FUNCTION_BLOCK FB_SimulatedScale EXTENDS FB_ComponentBase IMPLEMENTS I_Scale
VAR_INPUT
END_VAR
VAR_OUTPUT
END_VAR
VAR
END_VAR

{warning 'Add method implementation '}
METHOD CyclicLogic
END_METHOD

{warning 'Add method implementation '}
METHOD Tare
END_METHOD

{warning 'Add property implementation'}
PROPERTY Weight : LREAL
GET
END_GET
SET
END_SET
END_PROPERTY

END_FUNCTION_BLOCK

(* stored: Version 1.1.0.1
   POU FB_SimulatedScale: Id {4daf688a-6a4f-43ef-98c9-d12265253220}, SpecialFunc None
   Method CyclicLogic: Id {8eb76a38-87f9-4e72-b49b-7fc2f5b7cd9a}
   Method Tare: Id {bd2a2a9b-4af6-4061-af68-9126198b4727}
   Property Weight: Id {1f8d0437-5694-4f7a-9da5-16a41e9d4959}
   Get Get: Id {5b4e41ee-cdee-4f21-8763-6190b3e04481}
   Set Set: Id {6fbe45c1-3ab9-4af4-a5ed-2904847823fc} *)
